(* CoDeSys 2.3 export: FX_PORTE_VITESSE.EXP *)

(* POU Simulation_Visuelle/FX_Porte_Vitesse, ST *)
FUNCTION FX_Porte_Vitesse : REAL
VAR_INPUT
	PosXPorte: INT;
END_VAR
VAR
	VarLocalA: REAL;
	ValXLocal: REAL;
END_VAR
(*Cette fonction retourne la position X de la porte gauche en fonction de la position X de la porte droite*)
(* Elle permet une exacte synchronisation des deux portes*)
VarLocalA:=-(59.0/71.0);
ValXLocal:= INT_TO_REAL(PosXPorte);
FX_Porte_Vitesse:=(VarLocalA)*(ValXLocal);
END_FUNCTION
